// TIA Portal V17 export
// export: Created 2024-11-22T10:16:34.1632213Z, ExportSetting WithDefaults, DisplayName Totally Integrated Automation Portal, DisplayVersion V17, DisplayName TIA Portal Openness, DisplayVersion V17, DisplayName TIA Portal Version Control Interface, DisplayVersion V17, DisplayName STEP 7 Professional, DisplayVersion V17, DisplayName STEP 7 Safety, DisplayVersion V17, DisplayName WinCC Professional, DisplayVersion V17
VAR_GLOBAL   // PLC tag table "UserDiag_Constants"
END_VAR
VAR_GLOBAL CONSTANT   // user constants
   USERDIAG_IOSYSTEM_1 : Int := 1;   // Index for first IO-System/DP-Mastersystem
   USERDIAG_DEVICES_PER_IO_SYSTEM_UPPER_LIM : Int := 5;   // Upper limit of devices/slaves per IO-System/DP-Mastersystem
   USERDIAG_SLOTS_PER_PLC_UPPER_LIM : Int := 9;   // max number of local modules
   USERDIAG_IO_SYSTEMS_UPPER_LIM : Int := 1;   // Upper limit of IO-Systems/DP-Mastersystems
   USERDIAG_DEVICES_PER_SCREEN_UPPER_LIM : Int := 5;   // Upper limit of devices per HMI screen
   USERDIAG_SLOTS_PER_SCREEN_UPPER_LIM : Int := 9;   // Upper limit of slots per HMI screen
   USERDIAG_SLOTS_PER_DEVICE_UPPER_LIM : Int := 9;   // max number of modules per device
END_VAR
